FUNCTION_BLOCK ADD_2 (* Calculate arithmetical sum of magnitude inputs (generic FB) *)
  (* Standard: 61131-3; Classification: standard arithmetic function; Description: Copyright (c) 2014 Profactor GmbH This program and the accompanying materials are made available under the terms of the Eclipse Public License 2.0 which is available at https://www.eclipse.org/legal/epl-2.0/ SPDX-License-Identifier: EPL-2.0 *)
  (* Version 1.0, 2014-10-11, Matthias Plasch, Profactor GmbH *)
  {SET_ATTRIBUTE(GenericClassName, 'GEN_ADD')}
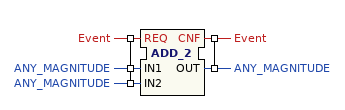
  EVENT_INPUT
    REQ WITH IN1, IN2; (* Normal Execution Request *)
  END_EVENT
  EVENT_OUTPUT
    CNF WITH OUT; (* Execution Confirmation *)
  END_EVENT
  VAR_INPUT
    IN1 : ANY_MAGNITUDE; (* ADD input 1 *)
    IN2 : ANY_MAGNITUDE; (* ADD input 2 *)
  END_VAR
  VAR_OUTPUT
    OUT : ANY_MAGNITUDE; (* ADD result *)
  END_VAR
END_FUNCTION_BLOCK
